PROGRAM P_Safety_Mapping
VAR
	fbF_Trig: F_TRIG;
END_VAR






//	GVL_PLC.bSafetySystemResetRequired := TRUE;


//IF GVL_Safe_IO.bAck_Error THEN
//	GVL_PLC.bSafetySystemResetRequired := FALSE;
//END_IF

//Comms to TwinSAFE
GVL_Safe_IO.bES_Restart_Local 		:= GVL_PLC.bLocalEstopRestart ;
GVL_Safe_IO.bAck_Error				:= GVL_PLC.bSafetyErrAckInput ;
//GVL_Safe_IO.bExternalEstopEn 		:= GVL_PLC.bExternalEstopEnInput;
//GVL_Safe_IO.bES_Restart_External	:= GVL_PLC.bExternalEstopRestart;


//Comms to Ethercat Slave Network

END_PROGRAM

(* stored: Version 1.1.0.1, ProductVersion 3.1.4022.3
   POU P_Safety_Mapping: Id {55c6d51b-2b55-49b8-ab39-0c19ab75e223}, SpecialFunc None *)
